// TIA Portal V20 export
ORGANIZATION_BLOCK "Main"   // OB1, LAD, ProgramCycle
TITLE = "Main Program Sweep (Cycle)"
{ S7_Optimized_Access := 'TRUE' }
// stored: SetENOAutomatically false
   VAR_INPUT
      Initial_Call : Bool;   // Initial call of this OB
      Remanence : Bool;   // =True, if remanent data are available
   END_VAR
   VAR CONSTANT
      Test_Station : SInt := 2;
      Total_Number_Test_Stations : SInt := 25;
   END_VAR
BEGIN

REGION Network 1: Digital Inputs
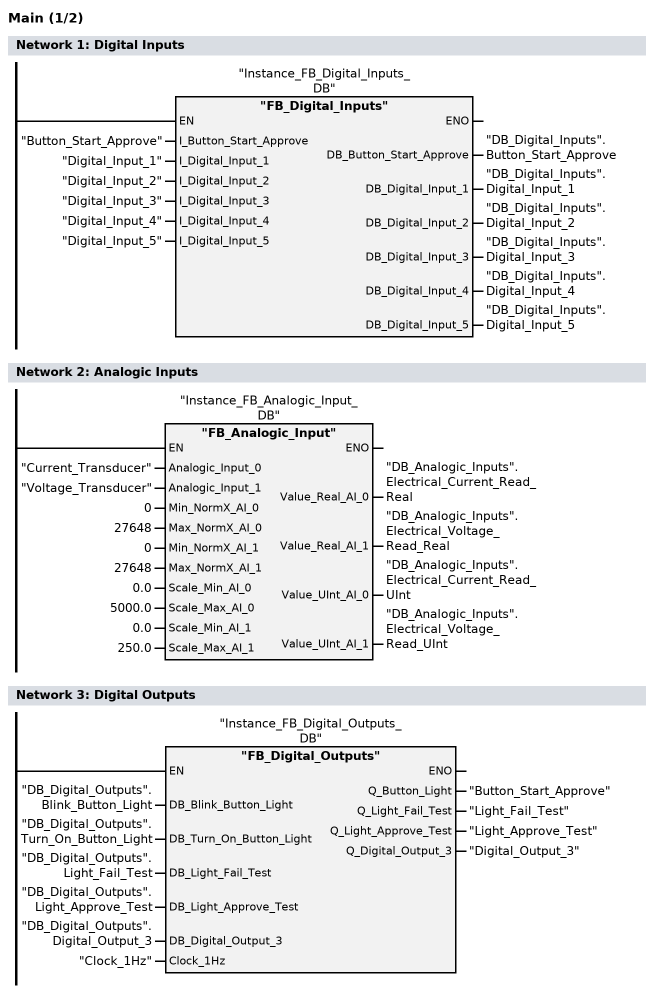
   RUNG wire#powerrail
      "Instance_FB_Digital_Inputs_DB"(I_Button_Start_Approve := "Button_Start_Approve", I_Digital_Input_1 := "Digital_Input_1", I_Digital_Input_2 := "Digital_Input_2", I_Digital_Input_3 := "Digital_Input_3", I_Digital_Input_4 := "Digital_Input_4", I_Digital_Input_5 := "Digital_Input_5", DB_Button_Start_Approve => "DB_Digital_Inputs".Button_Start_Approve, DB_Digital_Input_1 => "DB_Digital_Inputs".Digital_Input_1, DB_Digital_Input_2 => "DB_Digital_Inputs".Digital_Input_2, DB_Digital_Input_3 => "DB_Digital_Inputs".Digital_Input_3, DB_Digital_Input_4 => "DB_Digital_Inputs".Digital_Input_4, DB_Digital_Input_5 => "DB_Digital_Inputs".Digital_Input_5)
   END_RUNG
   // the same network as SCL:
   "Instance_FB_Digital_Inputs_DB"(I_Button_Start_Approve := "Button_Start_Approve",   // "FB_Digital_Inputs"
                           I_Digital_Input_1 := "Digital_Input_1",
                           I_Digital_Input_2 := "Digital_Input_2",
                           I_Digital_Input_3 := "Digital_Input_3",
                           I_Digital_Input_4 := "Digital_Input_4",
                           I_Digital_Input_5 := "Digital_Input_5",
                           DB_Button_Start_Approve => "DB_Digital_Inputs".Button_Start_Approve,
                           DB_Digital_Input_1 => "DB_Digital_Inputs".Digital_Input_1,
                           DB_Digital_Input_2 => "DB_Digital_Inputs".Digital_Input_2,
                           DB_Digital_Input_3 => "DB_Digital_Inputs".Digital_Input_3,
                           DB_Digital_Input_4 => "DB_Digital_Inputs".Digital_Input_4,
                           DB_Digital_Input_5 => "DB_Digital_Inputs".Digital_Input_5);
END_REGION

REGION Network 2: Analogic Inputs
   RUNG wire#powerrail
      "Instance_FB_Analogic_Input_DB"(Analogic_Input_0 := "Current_Transducer", Analogic_Input_1 := "Voltage_Transducer", Min_NormX_AI_0 := 0, Max_NormX_AI_0 := 27648, Min_NormX_AI_1 := 0, Max_NormX_AI_1 := 27648, Scale_Min_AI_0 := 0.0, Scale_Max_AI_0 := 5000.0, Scale_Min_AI_1 := 0.0, Scale_Max_AI_1 := 250.0, Value_Real_AI_0 => "DB_Analogic_Inputs".Electrical_Current_Read_Real, Value_Real_AI_1 => "DB_Analogic_Inputs".Electrical_Voltage_Read_Real, Value_UInt_AI_0 => "DB_Analogic_Inputs".Electrical_Current_Read_UInt, Value_UInt_AI_1 => "DB_Analogic_Inputs".Electrical_Voltage_Read_UInt)
   END_RUNG
   // the same network as SCL:
   "Instance_FB_Analogic_Input_DB"(Analogic_Input_0 := "Current_Transducer",   // "FB_Analogic_Input"
                           Analogic_Input_1 := "Voltage_Transducer",
                           Min_NormX_AI_0 := 0,
                           Max_NormX_AI_0 := 27648,
                           Min_NormX_AI_1 := 0,
                           Max_NormX_AI_1 := 27648,
                           Scale_Min_AI_0 := 0.0,
                           Scale_Max_AI_0 := 5000.0,
                           Scale_Min_AI_1 := 0.0,
                           Scale_Max_AI_1 := 250.0,
                           Value_Real_AI_0 => "DB_Analogic_Inputs".Electrical_Current_Read_Real,
                           Value_Real_AI_1 => "DB_Analogic_Inputs".Electrical_Voltage_Read_Real,
                           Value_UInt_AI_0 => "DB_Analogic_Inputs".Electrical_Current_Read_UInt,
                           Value_UInt_AI_1 => "DB_Analogic_Inputs".Electrical_Voltage_Read_UInt);
END_REGION

REGION Network 3: Digital Outputs
   RUNG wire#powerrail
      "Instance_FB_Digital_Outputs_DB"(DB_Blink_Button_Light := "DB_Digital_Outputs".Blink_Button_Light, DB_Turn_On_Button_Light := "DB_Digital_Outputs".Turn_On_Button_Light, DB_Light_Fail_Test := "DB_Digital_Outputs".Light_Fail_Test, DB_Light_Approve_Test := "DB_Digital_Outputs".Light_Approve_Test, DB_Digital_Output_3 := "DB_Digital_Outputs".Digital_Output_3, Clock_1Hz := "Clock_1Hz", Q_Button_Light => "Button_Start_Approve", Q_Light_Fail_Test => "Light_Fail_Test", Q_Light_Approve_Test => "Light_Approve_Test", Q_Digital_Output_3 => "Digital_Output_3")
   END_RUNG
   // the same network as SCL:
   "Instance_FB_Digital_Outputs_DB"(DB_Blink_Button_Light := "DB_Digital_Outputs".Blink_Button_Light,   // "FB_Digital_Outputs"
                           DB_Turn_On_Button_Light := "DB_Digital_Outputs".Turn_On_Button_Light,
                           DB_Light_Fail_Test := "DB_Digital_Outputs".Light_Fail_Test,
                           DB_Light_Approve_Test := "DB_Digital_Outputs".Light_Approve_Test,
                           DB_Digital_Output_3 := "DB_Digital_Outputs".Digital_Output_3,
                           Clock_1Hz := "Clock_1Hz",
                           Q_Button_Light => "Button_Start_Approve",
                           Q_Light_Fail_Test => "Light_Fail_Test",
                           Q_Light_Approve_Test => "Light_Approve_Test",
                           Q_Digital_Output_3 => "Digital_Output_3");
END_REGION

REGION Network 4: IO Device
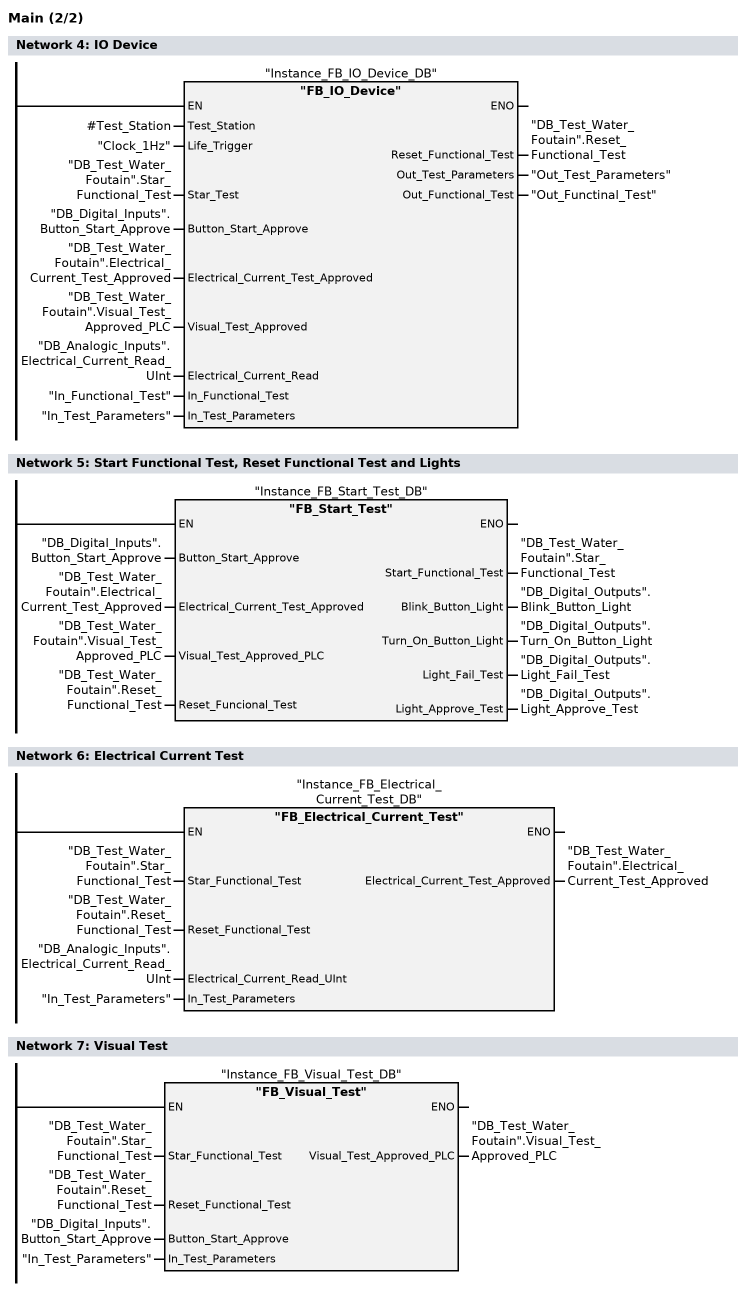
   RUNG wire#powerrail
      "Instance_FB_IO_Device_DB"(Test_Station := #Test_Station, Life_Trigger := "Clock_1Hz", Star_Test := "DB_Test_Water_Foutain".Star_Functional_Test, Button_Start_Approve := "DB_Digital_Inputs".Button_Start_Approve, Electrical_Current_Test_Approved := "DB_Test_Water_Foutain".Electrical_Current_Test_Approved, Visual_Test_Approved := "DB_Test_Water_Foutain".Visual_Test_Approved_PLC, Electrical_Current_Read := "DB_Analogic_Inputs".Electrical_Current_Read_UInt, In_Functional_Test := "In_Functional_Test", In_Test_Parameters := "In_Test_Parameters", Reset_Functional_Test => "DB_Test_Water_Foutain".Reset_Functional_Test, Out_Test_Parameters => "Out_Test_Parameters", Out_Functional_Test => "Out_Functinal_Test")
   END_RUNG
   // the same network as SCL:
   "Instance_FB_IO_Device_DB"(Test_Station := #Test_Station,   // "FB_IO_Device"
                           Life_Trigger := "Clock_1Hz",
                           Star_Test := "DB_Test_Water_Foutain".Star_Functional_Test,
                           Button_Start_Approve := "DB_Digital_Inputs".Button_Start_Approve,
                           Electrical_Current_Test_Approved := "DB_Test_Water_Foutain".Electrical_Current_Test_Approved,
                           Visual_Test_Approved := "DB_Test_Water_Foutain".Visual_Test_Approved_PLC,
                           Electrical_Current_Read := "DB_Analogic_Inputs".Electrical_Current_Read_UInt,
                           In_Functional_Test := "In_Functional_Test",
                           In_Test_Parameters := "In_Test_Parameters",
                           Reset_Functional_Test => "DB_Test_Water_Foutain".Reset_Functional_Test,
                           Out_Test_Parameters => "Out_Test_Parameters",
                           Out_Functional_Test => "Out_Functinal_Test");
END_REGION

REGION Network 5: Start Functional Test, Reset Functional Test and Lights
   RUNG wire#powerrail
      "Instance_FB_Start_Test_DB"(Button_Start_Approve := "DB_Digital_Inputs".Button_Start_Approve, Electrical_Current_Test_Approved := "DB_Test_Water_Foutain".Electrical_Current_Test_Approved, Visual_Test_Approved_PLC := "DB_Test_Water_Foutain".Visual_Test_Approved_PLC, Reset_Funcional_Test := "DB_Test_Water_Foutain".Reset_Functional_Test, Start_Functional_Test => "DB_Test_Water_Foutain".Star_Functional_Test, Blink_Button_Light => "DB_Digital_Outputs".Blink_Button_Light, Turn_On_Button_Light => "DB_Digital_Outputs".Turn_On_Button_Light, Light_Fail_Test => "DB_Digital_Outputs".Light_Fail_Test, Light_Approve_Test => "DB_Digital_Outputs".Light_Approve_Test)
   END_RUNG
   // the same network as SCL:
   "Instance_FB_Start_Test_DB"(Button_Start_Approve := "DB_Digital_Inputs".Button_Start_Approve,   // "FB_Start_Test"
                           Electrical_Current_Test_Approved := "DB_Test_Water_Foutain".Electrical_Current_Test_Approved,
                           Visual_Test_Approved_PLC := "DB_Test_Water_Foutain".Visual_Test_Approved_PLC,
                           Reset_Funcional_Test := "DB_Test_Water_Foutain".Reset_Functional_Test,
                           Start_Functional_Test => "DB_Test_Water_Foutain".Star_Functional_Test,
                           Blink_Button_Light => "DB_Digital_Outputs".Blink_Button_Light,
                           Turn_On_Button_Light => "DB_Digital_Outputs".Turn_On_Button_Light,
                           Light_Fail_Test => "DB_Digital_Outputs".Light_Fail_Test,
                           Light_Approve_Test => "DB_Digital_Outputs".Light_Approve_Test);
END_REGION

REGION Network 6: Electrical Current Test
   RUNG wire#powerrail
      "Instance_FB_Electrical_Current_Test_DB"(Star_Functional_Test := "DB_Test_Water_Foutain".Star_Functional_Test, Reset_Functional_Test := "DB_Test_Water_Foutain".Reset_Functional_Test, Electrical_Current_Read_UInt := "DB_Analogic_Inputs".Electrical_Current_Read_UInt, In_Test_Parameters := "In_Test_Parameters", Electrical_Current_Test_Approved => "DB_Test_Water_Foutain".Electrical_Current_Test_Approved)
   END_RUNG
   // the same network as SCL:
   "Instance_FB_Electrical_Current_Test_DB"(Star_Functional_Test := "DB_Test_Water_Foutain".Star_Functional_Test,   // "FB_Electrical_Current_Test"
                           Reset_Functional_Test := "DB_Test_Water_Foutain".Reset_Functional_Test,
                           Electrical_Current_Read_UInt := "DB_Analogic_Inputs".Electrical_Current_Read_UInt,
                           In_Test_Parameters := "In_Test_Parameters",
                           Electrical_Current_Test_Approved => "DB_Test_Water_Foutain".Electrical_Current_Test_Approved);
END_REGION

REGION Network 7: Visual Test
   RUNG wire#powerrail
      "Instance_FB_Visual_Test_DB"(Star_Functional_Test := "DB_Test_Water_Foutain".Star_Functional_Test, Reset_Functional_Test := "DB_Test_Water_Foutain".Reset_Functional_Test, Button_Start_Approve := "DB_Digital_Inputs".Button_Start_Approve, In_Test_Parameters := "In_Test_Parameters", Visual_Test_Approved_PLC => "DB_Test_Water_Foutain".Visual_Test_Approved_PLC)
   END_RUNG
   // the same network as SCL:
   "Instance_FB_Visual_Test_DB"(Star_Functional_Test := "DB_Test_Water_Foutain".Star_Functional_Test,   // "FB_Visual_Test"
                           Reset_Functional_Test := "DB_Test_Water_Foutain".Reset_Functional_Test,
                           Button_Start_Approve := "DB_Digital_Inputs".Button_Start_Approve,
                           In_Test_Parameters := "In_Test_Parameters",
                           Visual_Test_Approved_PLC => "DB_Test_Water_Foutain".Visual_Test_Approved_PLC);
END_REGION
END_ORGANIZATION_BLOCK
